{attribute 'GeneratedUsingTerminal: EK1960-2600-0021'}
{attribute addProperty BoxType "EK1960-2600-0021"}
{attribute addProperty Id "FSOEAT %I*FSOE_E251F24448"}
{attribute addProperty CRC "2717131454"}
{attribute addProperty Size "48"}
TYPE FSoE_Inputs_A1F422BE :
STRUCT
	{attribute addProperty Name "FSOE"}
	FSOE AT %I* : FSOE_E251F244;
END_STRUCT
END_TYPE

(* stored: Version 1.2.0.0, ProductVersion 3.1.4024.9
   DUT FSoE_Inputs_A1F422BE: Id {7b561110-6f68-4451-b3cd-b780ae3dee90} *)
